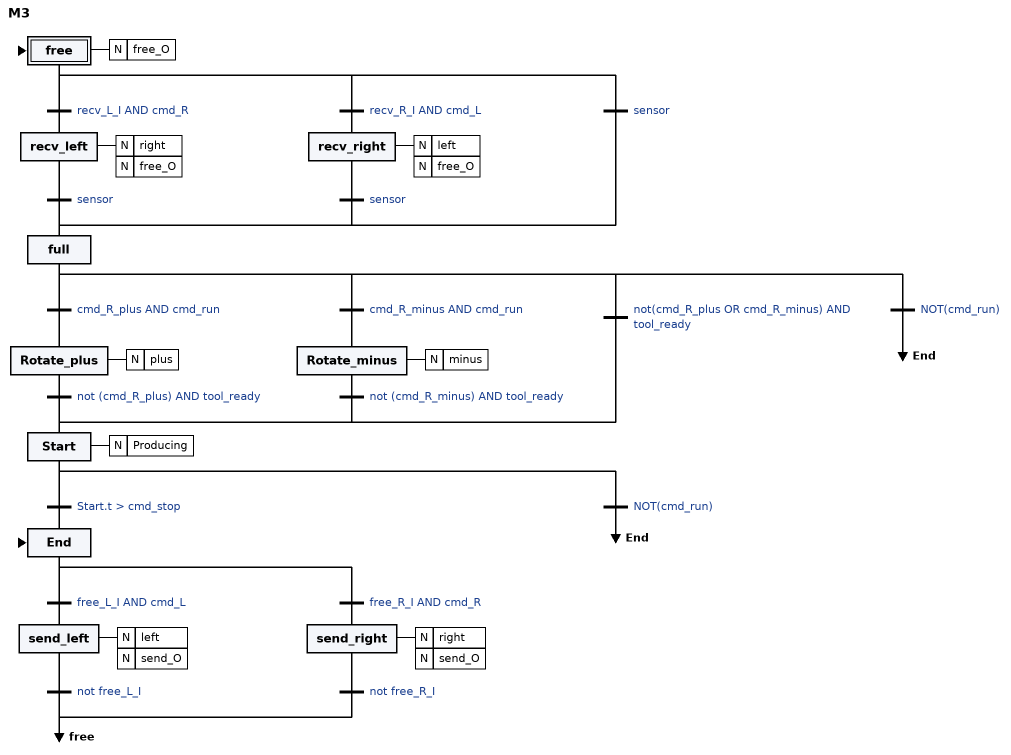
INITIAL_STEP free:
    free_O(N);
END_STEP
TRANSITION FROM free TO recv_left
    := recv_L_I AND cmd_R;
END_TRANSITION
STEP recv_left:
    right(N);
    free_O(N);
END_STEP
TRANSITION FROM recv_left TO full
    := sensor;
END_TRANSITION
TRANSITION FROM free TO recv_right
    := recv_R_I AND cmd_L;
END_TRANSITION
STEP recv_right:
    left(N);
    free_O(N);
END_STEP
TRANSITION FROM recv_right TO full
    := sensor;
END_TRANSITION
TRANSITION FROM free TO full
    := sensor;
END_TRANSITION
STEP full:
END_STEP
TRANSITION FROM full TO Rotate_plus
    := cmd_R_plus AND cmd_run;
END_TRANSITION
STEP Rotate_plus:
    plus(N);
END_STEP
TRANSITION FROM Rotate_plus TO Start
    := not (cmd_R_plus) AND tool_ready;
END_TRANSITION
TRANSITION FROM full TO Rotate_minus
    := cmd_R_minus AND cmd_run;
END_TRANSITION
STEP Rotate_minus:
    minus(N);
END_STEP
TRANSITION FROM Rotate_minus TO Start
    := not (cmd_R_minus) AND tool_ready;
END_TRANSITION
TRANSITION FROM full TO Start
    := not(cmd_R_plus OR cmd_R_minus) AND tool_ready;
END_TRANSITION
TRANSITION FROM full TO End
    := NOT(cmd_run);
END_TRANSITION
STEP Start:
    Producing(N);
END_STEP
TRANSITION FROM Start TO End
    := Start.t > cmd_stop;
END_TRANSITION
TRANSITION FROM Start TO End
    := NOT(cmd_run);
END_TRANSITION
STEP End:
END_STEP
TRANSITION FROM End TO send_left
    := free_L_I AND cmd_L;
END_TRANSITION
STEP send_left:
    left(N);
    send_O(N);
END_STEP
TRANSITION FROM send_left TO free
    := not free_L_I;
END_TRANSITION
TRANSITION FROM End TO send_right
    := free_R_I AND cmd_R;
END_TRANSITION
STEP send_right:
    right(N);
    send_O(N);
END_STEP
TRANSITION FROM send_right TO free
    := not free_R_I;
END_TRANSITION

END_FUNCTION_BLOCK

// Device/Application/T_Lin_Psh_Up
FUNCTION_BLOCK T_Lin_Psh_Up
VAR_INPUT
	sensor: BOOL;
	free_L_I: BOOL;
	free_R_I: BOOL;
	recv_L_I: BOOL;
	recv_R_I: BOOL;
	cmd_L:BOOL;
	cmd_R:BOOL;
	cmd_in: BOOL;
	contracted: BOOL;
	extended: BOOL;
	space_free: BOOL;
		
END_VAR
VAR_OUTPUT
	left : BOOL;
	right : BOOL;
	free_O: BOOL;
	send_O: BOOL;
	transl_R: BOOL;
	transl_L: BOOL;
END_VAR
VAR
END_VAR

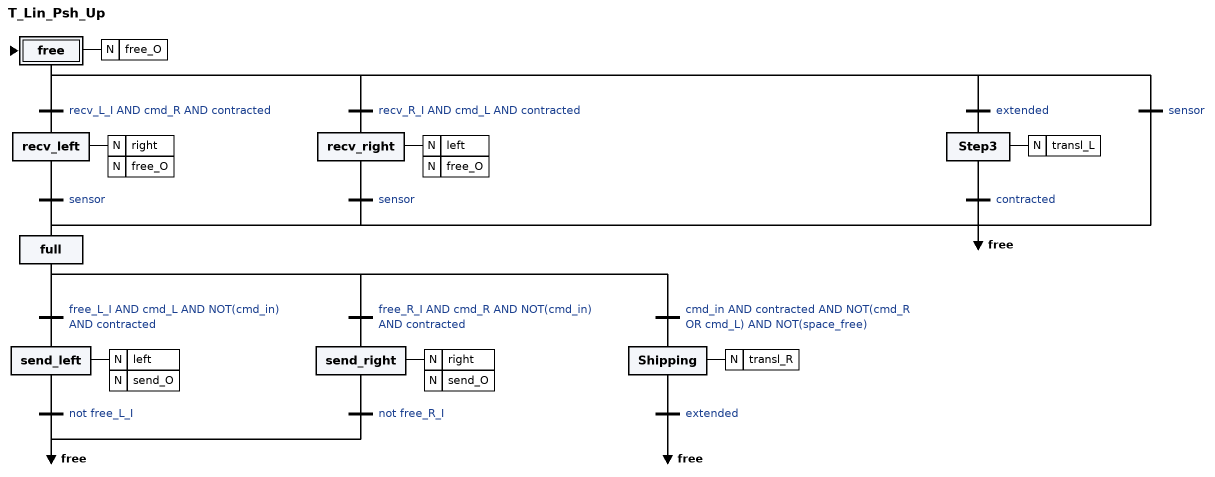
INITIAL_STEP free:
    free_O(N);
END_STEP
TRANSITION FROM free TO recv_left
    := recv_L_I AND cmd_R AND contracted;
END_TRANSITION
STEP recv_left:
    right(N);
    free_O(N);
END_STEP
TRANSITION FROM recv_left TO full
    := sensor;
END_TRANSITION
TRANSITION FROM free TO recv_right
    := recv_R_I AND cmd_L AND contracted;
END_TRANSITION
STEP recv_right:
    left(N);
    free_O(N);
END_STEP
TRANSITION FROM recv_right TO full
    := sensor;
END_TRANSITION
TRANSITION FROM free TO Step3
    := extended;
END_TRANSITION
STEP Step3:
    transl_L(N);
END_STEP
TRANSITION FROM Step3 TO free
    := contracted;
END_TRANSITION
TRANSITION FROM free TO full
    := sensor;
END_TRANSITION
STEP full:
END_STEP
TRANSITION FROM full TO send_left
    := free_L_I AND cmd_L AND NOT(cmd_in) AND contracted;
END_TRANSITION
STEP send_left:
    left(N);
    send_O(N);
END_STEP
TRANSITION FROM send_left TO free
    := not free_L_I;
END_TRANSITION
TRANSITION FROM full TO send_right
    := free_R_I AND cmd_R AND NOT(cmd_in) AND contracted;
END_TRANSITION
STEP send_right:
    right(N);
    send_O(N);
END_STEP
TRANSITION FROM send_right TO free
    := not free_R_I;
END_TRANSITION
TRANSITION FROM full TO Shipping
    := cmd_in AND contracted AND NOT(cmd_R OR cmd_L) AND NOT(space_free);
END_TRANSITION
STEP Shipping:
    transl_R(N);
END_STEP
TRANSITION FROM Shipping TO free
    := extended;
END_TRANSITION

END_FUNCTION_BLOCK

// Device/Application/T_Rot_Down
FUNCTION_BLOCK T_Rot_Down
VAR_INPUT
	sensor: BOOL;
	free_L_I: BOOL;
	free_R_I: BOOL;
	recv_L_I: BOOL;
	recv_R_I: BOOL;
	free_V_I: BOOL;
	recv_V_I: BOOL;
	cmd_L:BOOL;
	cmd_R:BOOL;
	cmd_Rotation_plus: BOOL;
	cmd_Rotation_minus: BOOL;
	horizontal: BOOL;
	vertical: BOOL;
	
END_VAR
VAR_OUTPUT
	left : BOOL;
	right : BOOL;
	rotate_plus : BOOL;
	rotate_minus : BOOL;
	free_O: BOOL;
	send_O: BOOL;
END_VAR
VAR
END_VAR

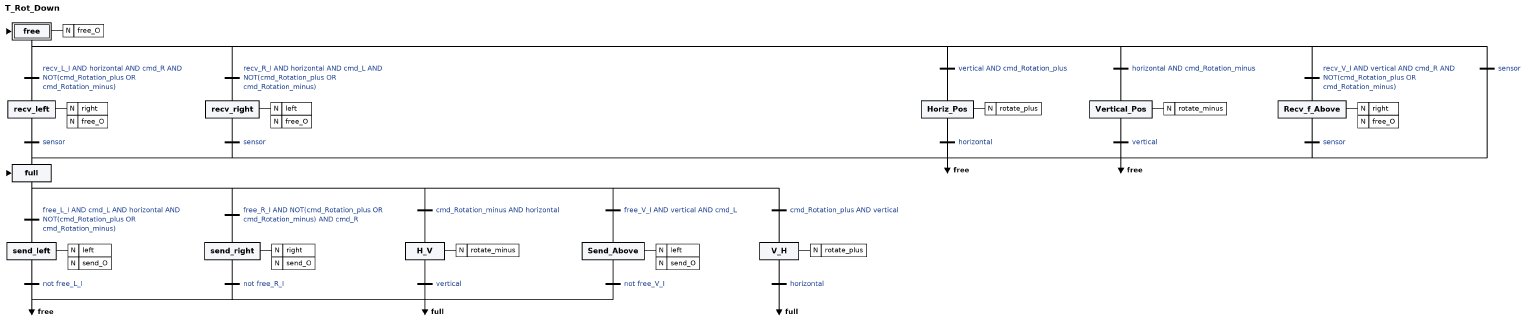
INITIAL_STEP free:
    free_O(N);
END_STEP
TRANSITION FROM free TO recv_left
    := recv_L_I AND horizontal AND cmd_R AND NOT(cmd_Rotation_plus OR cmd_Rotation_minus);
END_TRANSITION
STEP recv_left:
    right(N);
    free_O(N);
END_STEP
TRANSITION FROM recv_left TO full
    := sensor;
END_TRANSITION
TRANSITION FROM free TO recv_right
    := recv_R_I AND horizontal AND cmd_L AND NOT(cmd_Rotation_plus OR cmd_Rotation_minus);
END_TRANSITION
STEP recv_right:
    left(N);
    free_O(N);
END_STEP
TRANSITION FROM recv_right TO full
    := sensor;
END_TRANSITION
TRANSITION FROM free TO Horiz_Pos
    := vertical AND cmd_Rotation_plus;
END_TRANSITION
STEP Horiz_Pos:
    rotate_plus(N);
END_STEP
TRANSITION FROM Horiz_Pos TO free
    := horizontal;
END_TRANSITION
TRANSITION FROM free TO Vertical_Pos
    := horizontal AND cmd_Rotation_minus;
END_TRANSITION
STEP Vertical_Pos:
    rotate_minus(N);
END_STEP
TRANSITION FROM Vertical_Pos TO free
    := vertical;
END_TRANSITION
TRANSITION FROM free TO Recv_f_Above
    := recv_V_I AND vertical AND cmd_R AND NOT(cmd_Rotation_plus OR cmd_Rotation_minus);
END_TRANSITION
STEP Recv_f_Above:
    right(N);
    free_O(N);
END_STEP
TRANSITION FROM Recv_f_Above TO full
    := sensor;
END_TRANSITION
TRANSITION FROM free TO full
    := sensor;
END_TRANSITION
STEP full:
END_STEP
TRANSITION FROM full TO send_left
    := free_L_I AND cmd_L AND horizontal AND NOT(cmd_Rotation_plus OR cmd_Rotation_minus);
END_TRANSITION
STEP send_left:
    left(N);
    send_O(N);
END_STEP
TRANSITION FROM send_left TO free
    := not free_L_I;
END_TRANSITION
TRANSITION FROM full TO send_right
    := free_R_I AND NOT(cmd_Rotation_plus OR cmd_Rotation_minus) AND cmd_R;
END_TRANSITION
STEP send_right:
    right(N);
    send_O(N);
END_STEP
TRANSITION FROM send_right TO free
    := not free_R_I;
END_TRANSITION
TRANSITION FROM full TO H_V
    := cmd_Rotation_minus AND horizontal;
END_TRANSITION
STEP H_V:
    rotate_minus(N);
END_STEP
TRANSITION FROM H_V TO full
    := vertical;
END_TRANSITION
TRANSITION FROM full TO Send_Above
    := free_V_I AND vertical AND cmd_L;
END_TRANSITION
STEP Send_Above:
    left(N);
    send_O(N);
END_STEP
TRANSITION FROM Send_Above TO free
    := not free_V_I;
END_TRANSITION
TRANSITION FROM full TO V_H
    := cmd_Rotation_plus AND vertical;
END_TRANSITION
STEP V_H:
    rotate_plus(N);
END_STEP
TRANSITION FROM V_H TO full
    := horizontal;
END_TRANSITION

END_FUNCTION_BLOCK

// Device/Application/T_WH_in
FUNCTION_BLOCK T_WH_in
VAR_INPUT
	WH_Piece_Number: UINT;
	sensor: BOOL;
	free_R_I: BOOL;
	recv_R_I: BOOL;
	free_L_I: BOOL;
	cmd_R:BOOL;
	cmd_L:BOOL;
			
END_VAR
VAR_OUTPUT
	right : BOOL;
	left : BOOL;
	free_O: BOOL;
	send_O: BOOL;
	IN: BOOL;
END_VAR
VAR
END_VAR

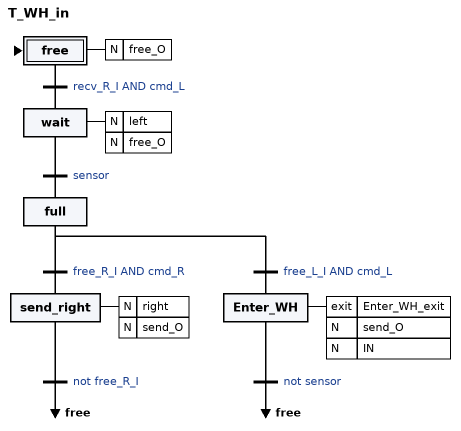
INITIAL_STEP free:
    free_O(N);
END_STEP
TRANSITION FROM free TO wait
    := recv_R_I AND cmd_L;
END_TRANSITION
STEP wait:
    left(N);
    free_O(N);
END_STEP
TRANSITION FROM wait TO full
    := sensor;
END_TRANSITION
STEP full:
END_STEP
TRANSITION FROM full TO send_right
    := free_R_I AND cmd_R;
END_TRANSITION
STEP send_right:
    right(N);
    send_O(N);
END_STEP
TRANSITION FROM send_right TO free
    := not free_R_I;
END_TRANSITION
TRANSITION FROM full TO Enter_WH
    := free_L_I AND cmd_L;
END_TRANSITION
STEP Enter_WH:
    Enter_WH_exit(P0);  // exit action
    send_O(N);
    IN(N);
END_STEP
TRANSITION FROM Enter_WH TO free
    := not sensor;
END_TRANSITION

ACTION Enter_WH_exit:
WH_Piece_Number:=WH_Piece_Number+1;
END_ACTION

END_FUNCTION_BLOCK

// Device/Application/T_Transl_Up
FUNCTION_BLOCK T_Transl_Up
VAR_INPUT
	sensor: BOOL;
	free_M3_I: BOOL;
	recv_M4_I: BOOL;
	free_M4_I: BOOL;
	recv_M3_I: BOOL;
	free_V_I: BOOL;
	recv_V_I: BOOL;
	cmd_MR: BOOL;
	cmd_ML: BOOL;
	vertical: BOOL;
	RIGHT_SIDE: BOOL;
	LEFT_SIDE: BOOL;
	cmd_R: BOOL;
	cmd_L: BOOL;
	
END_VAR
VAR_OUTPUT
	left : BOOL;
	right : BOOL;
	trans_left: BOOL;
	trans_right: BOOL;
	free_O: BOOL;
	send_O: BOOL;
END_VAR
VAR
	END_VAR

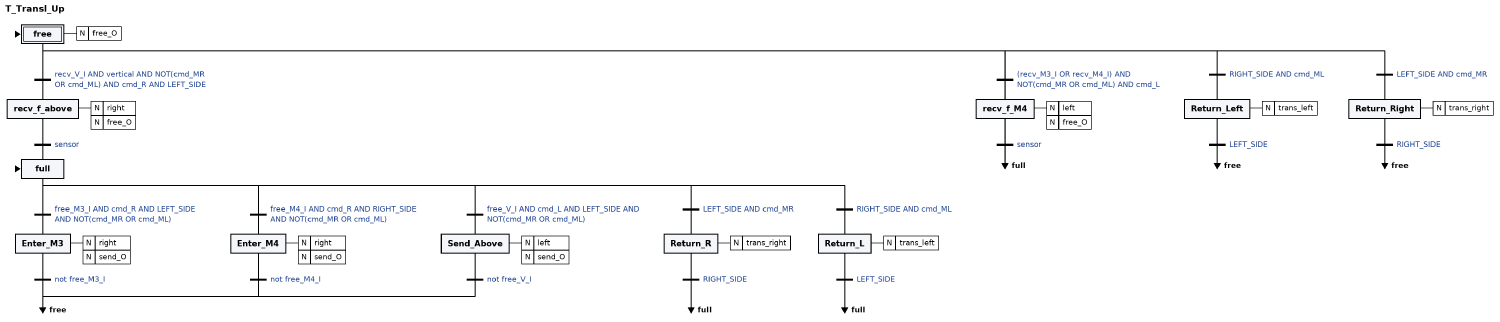
INITIAL_STEP free:
    free_O(N);
END_STEP
TRANSITION FROM free TO recv_f_above
    := recv_V_I AND vertical AND NOT(cmd_MR OR cmd_ML) AND cmd_R AND LEFT_SIDE;
END_TRANSITION
STEP recv_f_above:
    right(N);
    free_O(N);
END_STEP
TRANSITION FROM recv_f_above TO full
    := sensor;
END_TRANSITION
TRANSITION FROM free TO recv_f_M4
    := (recv_M3_I OR recv_M4_I) AND NOT(cmd_MR OR cmd_ML) AND cmd_L;
END_TRANSITION
STEP recv_f_M4:
    left(N);
    free_O(N);
END_STEP
TRANSITION FROM recv_f_M4 TO full
    := sensor;
END_TRANSITION
TRANSITION FROM free TO Return_Left
    := RIGHT_SIDE AND cmd_ML;
END_TRANSITION
STEP Return_Left:
    trans_left(N);
END_STEP
TRANSITION FROM Return_Left TO free
    := LEFT_SIDE;
END_TRANSITION
TRANSITION FROM free TO Return_Right
    := LEFT_SIDE AND cmd_MR;
END_TRANSITION
STEP Return_Right:
    trans_right(N);
END_STEP
TRANSITION FROM Return_Right TO free
    := RIGHT_SIDE;
END_TRANSITION
STEP full:
END_STEP
TRANSITION FROM full TO Enter_M3
    := free_M3_I AND cmd_R AND LEFT_SIDE AND NOT(cmd_MR OR cmd_ML);
END_TRANSITION
STEP Enter_M3:
    right(N);
    send_O(N);
END_STEP
TRANSITION FROM Enter_M3 TO free
    := not free_M3_I;
END_TRANSITION
TRANSITION FROM full TO Enter_M4
    := free_M4_I AND cmd_R AND RIGHT_SIDE AND NOT(cmd_MR OR cmd_ML);
END_TRANSITION
STEP Enter_M4:
    right(N);
    send_O(N);
END_STEP
TRANSITION FROM Enter_M4 TO free
    := not free_M4_I;
END_TRANSITION
TRANSITION FROM full TO Send_Above
    := free_V_I AND cmd_L AND LEFT_SIDE AND NOT(cmd_MR OR cmd_ML);
END_TRANSITION
STEP Send_Above:
    left(N);
    send_O(N);
END_STEP
TRANSITION FROM Send_Above TO free
    := not free_V_I;
END_TRANSITION
TRANSITION FROM full TO Return_R
    := LEFT_SIDE AND cmd_MR;
END_TRANSITION
STEP Return_R:
    trans_right(N);
END_STEP
TRANSITION FROM Return_R TO full
    := RIGHT_SIDE;
END_TRANSITION
TRANSITION FROM full TO Return_L
    := RIGHT_SIDE AND cmd_ML;
END_TRANSITION
STEP Return_L:
    trans_left(N);
END_STEP
TRANSITION FROM Return_L TO full
    := LEFT_SIDE;
END_TRANSITION

END_FUNCTION_BLOCK

// Device/Application/T_WH_out
FUNCTION_BLOCK T_WH_out
VAR_INPUT
	PieceToRemove: BYTE;
	sensor: BOOL;
	free_R_I: BOOL;
	cmd_R:BOOL;
			
END_VAR
VAR_OUTPUT
	right : BOOL;
	free_O: BOOL;
	send_O: BOOL;
END_VAR
VAR
END_VAR

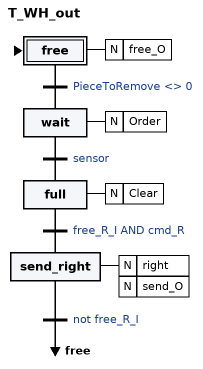
INITIAL_STEP free:
    free_O(N);
END_STEP
TRANSITION FROM free TO wait
    := PieceToRemove <> 0;
END_TRANSITION
STEP wait:
    Order(N);
END_STEP
TRANSITION FROM wait TO full
    := sensor;
END_TRANSITION
STEP full:
    Clear(N);
END_STEP
TRANSITION FROM full TO send_right
    := free_R_I AND cmd_R;
END_TRANSITION
STEP send_right:
    right(N);
    send_O(N);
END_STEP
TRANSITION FROM send_right TO free
    := not free_R_I;
END_TRANSITION

ACTION Clear:
GVL.R0:=0;
END_ACTION

ACTION Order:
GVL.R0:=PieceToRemove;
END_ACTION

END_FUNCTION_BLOCK

// Device/Application/T_Transl_Down
FUNCTION_BLOCK T_Transl_Down
VAR_INPUT
	sensor: BOOL;
	free_M3_I: BOOL;
	recv_M4_I: BOOL;
	free_M4_I: BOOL;
	recv_M3_I: BOOL;
	free_V_I: BOOL;
	recv_V_I: BOOL;
	cmd_MR: BOOL;
	cmd_ML: BOOL;
	vertical: BOOL;
	RIGHT_SIDE: BOOL;
	LEFT_SIDE: BOOL;
	cmd_R: BOOL;
	cmd_L: BOOL;
	
END_VAR
VAR_OUTPUT
	left : BOOL;
	right : BOOL;
	trans_left: BOOL;
	trans_right: BOOL;
	free_O: BOOL;
	send_O: BOOL;
END_VAR
VAR
	END_VAR

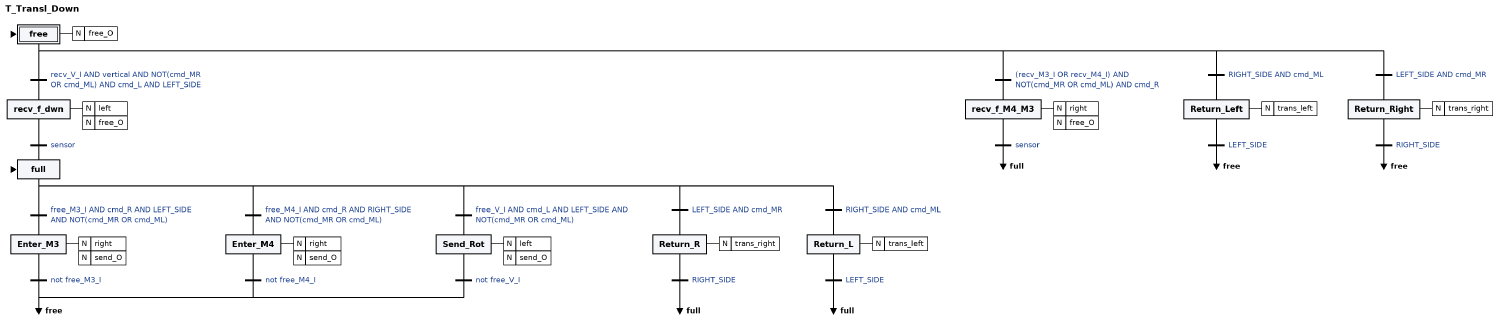
INITIAL_STEP free:
    free_O(N);
END_STEP
TRANSITION FROM free TO recv_f_dwn
    := recv_V_I AND vertical AND NOT(cmd_MR OR cmd_ML) AND cmd_L AND LEFT_SIDE;
END_TRANSITION
STEP recv_f_dwn:
    left(N);
    free_O(N);
END_STEP
TRANSITION FROM recv_f_dwn TO full
    := sensor;
END_TRANSITION
TRANSITION FROM free TO recv_f_M4_M3
    := (recv_M3_I OR recv_M4_I) AND NOT(cmd_MR OR cmd_ML) AND cmd_R;
END_TRANSITION
STEP recv_f_M4_M3:
    right(N);
    free_O(N);
END_STEP
TRANSITION FROM recv_f_M4_M3 TO full
    := sensor;
END_TRANSITION
TRANSITION FROM free TO Return_Left
    := RIGHT_SIDE AND cmd_ML;
END_TRANSITION
STEP Return_Left:
    trans_left(N);
END_STEP
TRANSITION FROM Return_Left TO free
    := LEFT_SIDE;
END_TRANSITION
TRANSITION FROM free TO Return_Right
    := LEFT_SIDE AND cmd_MR;
END_TRANSITION
STEP Return_Right:
    trans_right(N);
END_STEP
TRANSITION FROM Return_Right TO free
    := RIGHT_SIDE;
END_TRANSITION
STEP full:
END_STEP
TRANSITION FROM full TO Enter_M3
    := free_M3_I AND cmd_R AND LEFT_SIDE AND NOT(cmd_MR OR cmd_ML);
END_TRANSITION
STEP Enter_M3:
    right(N);
    send_O(N);
END_STEP
TRANSITION FROM Enter_M3 TO free
    := not free_M3_I;
END_TRANSITION
TRANSITION FROM full TO Enter_M4
    := free_M4_I AND cmd_R AND RIGHT_SIDE AND NOT(cmd_MR OR cmd_ML);
END_TRANSITION
STEP Enter_M4:
    right(N);
    send_O(N);
END_STEP
TRANSITION FROM Enter_M4 TO free
    := not free_M4_I;
END_TRANSITION
TRANSITION FROM full TO Send_Rot
    := free_V_I AND cmd_L AND LEFT_SIDE AND NOT(cmd_MR OR cmd_ML);
END_TRANSITION
STEP Send_Rot:
    left(N);
    send_O(N);
END_STEP
TRANSITION FROM Send_Rot TO free
    := not free_V_I;
END_TRANSITION
TRANSITION FROM full TO Return_R
    := LEFT_SIDE AND cmd_MR;
END_TRANSITION
STEP Return_R:
    trans_right(N);
END_STEP
TRANSITION FROM Return_R TO full
    := RIGHT_SIDE;
END_TRANSITION
TRANSITION FROM full TO Return_L
    := RIGHT_SIDE AND cmd_ML;
END_TRANSITION
STEP Return_L:
    trans_left(N);
END_STEP
TRANSITION FROM Return_L TO full
    := LEFT_SIDE;
END_TRANSITION

END_FUNCTION_BLOCK

// Device/Application/TimeMeas
PROGRAM TimeMeas
VAR
	Tempo: UDINT;
	TempoS: UDINT;
END_VAR

//Tempo := Systime().ClockTime;
Tempo:=SystimeCore.SysTimeGetMs();
TempoS:=Tempo/1000;

END_PROGRAM

// Device/Application/Tool_Counter
FUNCTION_BLOCK Tool_Counter
VAR_INPUT
	State: BYTE;
	END_VAR
VAR_OUTPUT
END_VAR
VAR
END_VAR

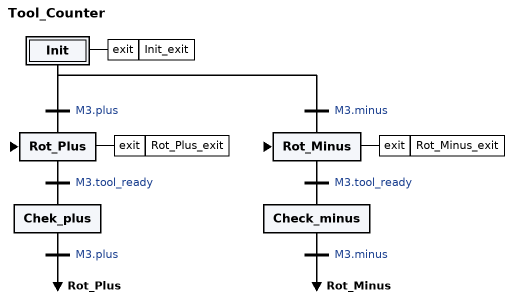
INITIAL_STEP Init:
    Init_exit(P0);  // exit action
END_STEP
TRANSITION FROM Init TO Rot_Plus
    := M3.plus;
END_TRANSITION
STEP Rot_Plus:
    Rot_Plus_exit(P0);  // exit action
END_STEP
TRANSITION FROM Rot_Plus TO Chek_plus
    := M3.tool_ready;
END_TRANSITION
STEP Chek_plus:
END_STEP
TRANSITION FROM Chek_plus TO Rot_Plus
    := M3.plus;
END_TRANSITION
TRANSITION FROM Init TO Rot_Minus
    := M3.minus;
END_TRANSITION
STEP Rot_Minus:
    Rot_Minus_exit(P0);  // exit action
END_STEP
TRANSITION FROM Rot_Minus TO Check_minus
    := M3.tool_ready;
END_TRANSITION
STEP Check_minus:
END_STEP
TRANSITION FROM Check_minus TO Rot_Minus
    := M3.minus;
END_TRANSITION

ACTION Init_exit:
State:=1;
END_ACTION

ACTION Rot_Minus_exit:
IF(State = 1)THEN State := 3;
END_IF
IF(State = 2)THEN State := 1;
END_IF
IF(State = 3)THEN State := 2;
END_IF
END_ACTION

ACTION Rot_Plus_exit:
IF(State = 1)THEN State := 2;
END_IF
IF(State = 2)THEN State := 3;
END_IF
IF(State = 3)THEN State := 1;
END_IF
END_ACTION

END_FUNCTION_BLOCK
